FUNCTION TryConvert_ULINT_TO_LWORD : BOOL
VAR_INPUT
	in : ULINT;
	out : REFERENCE TO LWORD;
END_VAR

out := ULINT_TO_LWORD(in);
TryConvert_ULINT_TO_LWORD := TRUE;

END_FUNCTION

(* stored: Version 1.1.0.1, ProductVersion 3.1.4024.12
   POU TryConvert_ULINT_TO_LWORD: Id {2f51f36d-9088-42f0-a734-524fc4797179}, SpecialFunc None *)
